TYPE SC_BUSY_SecondFloor :
(
	eSecondFloorStart := 0,
	eActivateTurn,
	eActivateBeltForw,
	eWaitForPackages,
	ePushPackages,
	eRetractPusher,
	eClamp,
	eRetractClamper,
	eWaitForPallet,
	eOpenPlate,
	eClosePlate,
	eElevatorUp,
	eElevatorDown,
	eStartChains,
	eStopChains,
	eWaitForFirstFloor,
	eSyncWithFirstFloor,
	eSecondFloorDone
);
END_TYPE

(* stored: Version 1.1.0.1, ProductVersion 3.1.4024.2
   DUT SC_BUSY_SecondFloor: Id {c088b052-b956-447b-9fd2-097aec83e820} *)
